Fanuc KAREL source: kt00330.KL

-- PROVISIONAL review KL for V940-1; original PC SHA256 586ea2900547df78afed2559b39a7f14e46145ae75481149b3c6c6e75504f726
-- Incomplete behavior may be omitted. Consult companion uncertainty JSON. Do not deploy.
PROGRAM KT00330
%NOLOCKGROUP
VAR
  I1 : INTEGER
  R2 : REAL
  OUT : BOOLEAN
BEGIN
  -- V9_ZERO_TABLE_METADATA_HINT layout=0001; no indexed target words; source/name/runtime held
  -- UNRESOLVED_PC offsets 5-16; opcodes 2E,23
  -- UNRESOLVED_PC offsets 21-32; opcodes 2E,23
  -- UNRESOLVED_PC offsets 37-59; opcodes 21,21,29,64,29,6F,23
  -- UNRESOLVED_PC offsets 64-68; opcodes 7F
END KT00330
